// TIA Portal V17 export
// export: Created 2024-01-30T08:49:12.5559508Z, ExportSetting WithDefaults, DisplayName Totally Integrated Automation Portal, DisplayVersion V17 Update 6, DisplayName TIA Portal Openness, DisplayVersion V17 Update 6, DisplayName TIA Portal Version Control Interface, DisplayVersion V17, DisplayName STEP 7 Professional, DisplayVersion V17 Update 6, DisplayName STEP 7 Safety, DisplayVersion V17 Update 6, DisplayName WinCC Advanced, DisplayVersion V17 Update 6
FUNCTION_BLOCK "Keyence_LJX8000_CTRL"   // FB14, LAD
{ S7_Optimized_Access := 'TRUE' }
VERSION : 0.1
// stored: AutoNumber true, IsIECCheckEnabled false, IsRetainMemResEnabled false, MemoryReserve 100, SetENOAutomatically false, UDAEnableTagReadback false
   VAR_INPUT
      PLC_IN_Bits : "UDT_LJ_X8000 --> PLC_Bits";
      PLC_IN_Bytes : "UDT_LJ_X8000 --> PLC_Bytes";
      RESET : Bool;
      CMD_NUMBER : DInt;
      PRG_NUMBER : DInt;
      CMD_REQ : Bool;
      TRIGGER : Bool;
      SD_CARD_NUM : DInt := 1;
   END_VAR
   VAR_OUTPUT
      ERROR : Bool;
      ACTIVE_CMD : DInt;
      ACTIVE_PRG : DInt;
      CMD_READY : Bool;
      HEAD_READY : Bool;
      HEAD_BUSY : Bool;
      SYSTEM_RUN : Bool;
      CMD_COMPLETE : Bool;
   END_VAR
   VAR_IN_OUT
      PLC_OUT_Bits : "UDT_PLC --> LJ_X8000_Bits";
      PLC_Out_Bytes : "UDT_PLC --> LJ_X8000_Bytes";
   END_VAR
   VAR
      ChangeToRun : Bool;
      ChangeToSetup : Bool;
   END_VAR
   VAR CONSTANT
      T1_Trigger : DInt := 1;
      R0_SwitchToRunMode : DInt := 8;
      S0_SwitchToSetupMode : DInt := 9;
      RS_Reset : DInt := 10;
      RB_Reboot : DInt := 11;
      SS_SaveProgram : DInt := 12;
      CE_ClearError : DInt := 13;
      VW_ChangeTheOperationScreen : DInt := 14;
      RM_ReadRunSetupMode : DInt := 16;
      PW_ChangeInspectionPrograms : DInt := 24;
      PR_ReadProgramSetting : DInt := 25;
      CTD_TriggerDelay : DInt := 34;
   END_VAR
BEGIN

REGION Network 1: Bit0
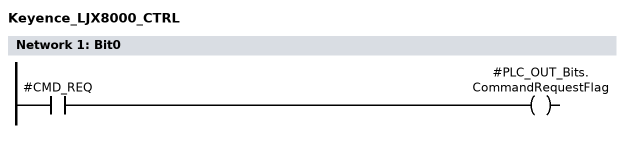
   RUNG wire#powerrail
      Contact( #CMD_REQ )
      Coil( #PLC_OUT_Bits.CommandRequestFlag )
   END_RUNG
   // the same network as SCL:
   #PLC_OUT_Bits.CommandRequestFlag := #CMD_REQ;
END_REGION

REGION Network 2 (SCL): Move data from PLC to Keyence
   #PLC_Out_Bytes.CommandNumber := #CMD_NUMBER;
   #PLC_Out_Bytes.ProgNumber := #PRG_NUMBER;
   #PLC_Out_Bytes.SDCardNumber := #SD_CARD_NUM;


   #PLC_OUT_Bits.ErrorResetRequestFlag := #RESET;
   #PLC_OUT_Bits.Trigger := #TRIGGER;


   #ACTIVE_CMD := #PLC_Out_Bytes.CommandNumber;
END_REGION

REGION Network 3 (SCL): Read data from Keyence
   #ERROR := #PLC_IN_Bits.Error;
   #CMD_READY := #PLC_IN_Bits.CommandReadFlag;
   #HEAD_READY := #PLC_IN_Bits.Ready;
   #HEAD_BUSY := #PLC_IN_Bits.Busy;
   #SYSTEM_RUN := #PLC_IN_Bits.Run;
   #CMD_COMPLETE := #PLC_IN_Bits.CommandCompleteFlag;



   // Bytes
   #ACTIVE_PRG := #PLC_IN_Bytes.CurrentPrgNumber;
END_REGION
END_FUNCTION_BLOCK
